{attribute 'linkalways'} 
{attribute 'no_explicit_call' := 'This FB is a CLASS and must be accessed using methods or properties'}
{attribute 'enable_dynamic_creation'}
FUNCTION_BLOCK AsyncResponseSessionData EXTENDS Disposable IMPLEMENTS I_AsyncResponseSessionData
VAR
	_suggestedRetryDelayInMs : UDINT;
	state : (PENDING, SUCCESS, SUCCESS_WITH_PAYLOAD, ERROR) := PENDING;
	errorCode : T_MAXSTRING;
	errorMessage : T_MAXSTRING;
	pData : POINTER TO BYTE;
	dataSize : UDINT;
END_VAR

METHOD PUBLIC CopyPayloadData
VAR_INPUT
	PayloadDataAddress : PVOID;
	PayloadDataSize : UDINT;
END_VAR
dataSize := PayloadDataSize;
pData := __NEW(BYTE, PayloadDataSize);
memcpy(pData,PayloadDataAddress,PayloadDataSize);
END_METHOD

METHOD PRIVATE DeletePayloadData
VAR_INPUT
END_VAR
IF pData = 0 THEN
	RETURN;
END_IF

__DELETE(pData);
dataSize := 0;
END_METHOD

METHOD PUBLIC Error
VAR_INPUT
	ErrorCode : T_MAXSTRING;
	Message : T_MAXSTRING;
END_VAR
IF state <> PENDING THEN
	RETURN;
END_IF

state := ERROR;
THIS^.errorCode := ErrorCode;
errorMessage := Message;
END_METHOD

METHOD FB_exit : BOOL
VAR_INPUT
	bInCopyCode : BOOL; // if TRUE, the exit method is called for exiting an instance that is copied afterwards (online change).
END_VAR
IF bInCopyCode THEN
	RETURN;
END_IF

DeletePayloadData();
END_METHOD

METHOD FB_init : BOOL
VAR_INPUT
	bInitRetains : BOOL; // if TRUE, the retain variables are initialized (warm start / cold start)
	bInCopyCode : BOOL;  // if TRUE, the instance afterwards gets moved into the copy code (online change)
	SuggestedRetryDelayInMs : UDINT;
END_VAR
_suggestedRetryDelayInMs := SuggestedRetryDelayInMs;
END_METHOD

PROPERTY PUBLIC IsPending : BOOL
GET
IsPending := state = PENDING;
END_GET
END_PROPERTY

METHOD PUBLIC Success
VAR_INPUT
END_VAR
IF state <> PENDING THEN
	RETURN;
END_IF

state := SUCCESS;
END_METHOD

METHOD PUBLIC SuccessWithPayload
VAR_INPUT
	PayloadDataAddress : PVOID;
	PayloadDataSize : UDINT;
END_VAR
IF state <> PENDING THEN
	RETURN;
END_IF

state := SUCCESS_WITH_PAYLOAD;
CopyPayloadData(PayloadDataAddress, PayloadDataSize);
END_METHOD

PROPERTY PUBLIC SuggestedRetryDelayInMs : UDINT
GET
SuggestedRetryDelayInMs := _suggestedRetryDelayInMs;
END_GET
SET // PUBLIC
_suggestedRetryDelayInMs := SuggestedRetryDelayInMs;
END_SET
END_PROPERTY

METHOD PUBLIC TryUpdateServerResponse : BOOL
VAR_INPUT
	Response : I_ServerResponse;
END_VAR
IF State = SUCCESS_WITH_PAYLOAD THEN
	Response.SuccessWithPayload(pData,dataSize);
	TryUpdateServerResponse := TRUE;
	RETURN;
END_IF

IF State = SUCCESS THEN
	Response.Success();
	TryUpdateServerResponse := TRUE;
	RETURN;
END_IF

IF state = ERROR THEN
	Response.Error(errorCode, errorMessage);
	TryUpdateServerResponse := TRUE;
	RETURN;
END_IF
END_METHOD

END_FUNCTION_BLOCK

(* stored: Version 1.1.0.1, ProductVersion 3.1.4026.13
   POU AsyncResponseSessionData: Id {0b8ed430-5a94-4796-b867-fe5806058bc5}, SpecialFunc None
   Folder Constructor: Id {6f42f4a9-b535-4973-9c62-6244f47596a3}
   Folder Destructor: Id {e41abfbe-c833-483c-92f1-81c6d7d7f286}
   Folder Private: Id {7ce13535-dc25-4f17-9951-0aa5f81cb2b6}
   Method CopyPayloadData: Id {37baa180-849b-46d5-a623-060e6ded8fc0}
   Method DeletePayloadData: Id {42be2907-e861-4d10-a4b5-c40a2b97a804}
   Method Error: Id {144bc9f0-3199-43a4-9154-95673c88ba76}
   Method FB_exit: Id {bc4d092b-2899-480a-bc7f-51f7fee36982}
   Method FB_init: Id {27f87d13-9903-48fc-8cff-7eca53b8e6d5}
   Property IsPending: Id {e08d9fad-bec8-4e32-95ab-a1cb4fcc9abe}
   Get Get: Id {b900a727-86a7-48c0-9cb8-f26a00a3183d}
   Method Success: Id {53d1f2b2-d75d-4cf7-ab0b-695555edeaaa}
   Method SuccessWithPayload: Id {26ccbc4d-1bd2-4e51-b563-1bfe2e48172f}
   Property SuggestedRetryDelayInMs: Id {8cb1d4ee-b5b9-45a6-83c9-9f2bf03df7c2}
   Get Get: Id {72f9dbe5-85f6-46e8-bfdb-69e04ad35781}
   Set Set: Id {6c6465cb-a651-4b7a-8d53-0295f21779e5}
   Method TryUpdateServerResponse: Id {42e916da-74e4-4d0b-9c4e-44edfd18f901} *)
